// TIA Portal V19 export
FUNCTION_BLOCK "Frequency"   // FB100, SCL
TITLE = Frequency
{ S7_Optimized_Access := 'TRUE' }
AUTHOR : Siemens
VERSION : 0.0.0.0
// Frequency (speed BeltLift)
// stored: IsIECCheckEnabled true, MemoryReserve 100, SetENOAutomatically true
   VAR_INPUT
      frequency { ExternalAccessible := 'False'; ExternalVisible := 'False'; ExternalWritable := 'False'} : Real := 10.0;   // Input in Hz
   END_VAR
   VAR_OUTPUT
      clock { ExternalAccessible := 'False'; ExternalVisible := 'False'; ExternalWritable := 'False'} : Bool;
      countdown { ExternalAccessible := 'False'; ExternalVisible := 'False'; ExternalWritable := 'False'} : Time;
      error { ExternalAccessible := 'False'; ExternalVisible := 'False'; ExternalWritable := 'False'} : Bool;
      status { ExternalAccessible := 'False'; ExternalVisible := 'False'; ExternalWritable := 'False'} : Word;
   END_VAR
   VAR
      instTofTimeOn { ExternalAccessible := 'False'; ExternalVisible := 'False'; ExternalWritable := 'False'; S7_SetPoint := 'True'} : TOF_TIME;
      instTofTimeOff { ExternalAccessible := 'False'; ExternalVisible := 'False'; ExternalWritable := 'False'; S7_SetPoint := 'True'} : TOF_TIME;
      statFrequencyMem { ExternalAccessible := 'False'; ExternalVisible := 'False'; ExternalWritable := 'False'} : Real;
      statTimeBase { ExternalAccessible := 'False'; ExternalVisible := 'False'; ExternalWritable := 'False'} : Time;
   END_VAR
   VAR CONSTANT
      MIN_FREQU : Real := 5.0;
      MAX_FREQU : Real := 10.0;
      FREQU_TO_LOW : Word := 16#8001;
      FREQU_TO_HIGH : Word := 16#8002;
   END_VAR
BEGIN
   //=============================================================================
   // Siemens AG
   // (c)Copyright 2015 All Rights Reserved
   //-----------------------------------------------------------------------------
   // Library:       LGF(Library General Functions)
   // Tested with:   CPU1212C DC/DC/DC FW:V4.1
   // Engineering:   TIA Portal V13 SP1 Upd 4
   // Restrictions:  -
   // Requirements:  PLC (S7-1200, S7-1500)
   // Functionality: Generates frequency signal
   //-----------------------------------------------------------------------------
   // Change log table:
   // Version  Date        Expert in charge                Changes applied
   // 01.00.00 21.07.2015  Siemens Industry Online Support First released version 
   //=============================================================================

   #error := FALSE;
   #status := 0;

   IF (#frequency <= 0.0)  // If input is <= 0.0 >> block is off // Wenn Eingang kleiner als 0.0 >> Baustein arbeitet nicht
   THEN
     #clock := FALSE;
     #countdown := t#0s;
   ELSE
     IF (#statFrequencyMem <> #frequency) // assign frequency one time   // Frequenz zuweisen
     THEN
       #statTimeBase := t#1000s / TRUNC(#frequency * 2000); // calculate time  //Zeit berechnen
       #statFrequencyMem := #frequency;
     END_IF;

     // TOF_off expired >> Start again // TOF_off abgelaufen starte von vorn
     #instTofTimeOn(IN := NOT #instTofTimeOff.Q,
                    PT := #statTimeBase);
     #countdown := #statTimeBase - #instTofTimeOn.ET;

     #instTofTimeOff(IN := #instTofTimeOn.Q,
                     PT := #statTimeBase);

     IF #countdown = t#0s THEN
       #countdown := #statTimeBase - #instTofTimeOff.ET;
     END_IF;

     #clock := #instTofTimeOn.Q; //assign ouptut // Frequenzausgang setzen   
   END_IF;

   //------------------------------------------------------------------------
   // Program for error message
   //------------------------------------------------------------------------
   IF (#frequency < #MIN_FREQU)
   THEN
     IF #status = 16#8002
     THEN
       #status := 0;
     ELSE
       #status := #FREQU_TO_LOW;
       #error := TRUE;
       RETURN;
     END_IF;
   END_IF;

   IF (#frequency > #MAX_FREQU)
   THEN
     IF #status = 16#8001
     THEN
       #status := 0;
     ELSE
       #status := #FREQU_TO_HIGH;
       #error := TRUE;
       RETURN;
     END_IF;
   END_IF;

   IF (#frequency = 10.0)
   THEN
     #status := 0;
     #error := 0;
     RETURN;
   END_IF;
END_FUNCTION_BLOCK
